FUNCTION_BLOCK ActivateTrackTask_TestSuite
VAR
	SetVelo AT%Q* : LREAL;
	AxisStatusFeedback AT%Q* : DWORD;
	stubAxis : AXIS_REF;
	stubTrack : XtsTrack('');
	testActivateTask : ActivateTrackTask := (AxisRef := stubAxis);
	TestSequence : INT;
	ThisTestSuite : TestSuite<TestSuiteParameter.MaxTestCount>('C:\ProgramData\Beckhoff\TwinCAT\3.1\Boot\ActiveTrack_Tests.xml') := (TestSuiteName := 'ActiveTrack Test Suite');
END_VAR

CASE TestSequence OF
	0: 
		SetVelo := 1.0;
		AxisStatusFeedback := 16#02100085;
		IF stubAxis.NcToPlc.SetVelo = 1.0 THEN
			TestSequence := 1;
		END_IF
	1:
		TaskRejectsCommandsWithNoAxis_Test();
		TaskRejectsDuplicateCommand_Test();
		TaskRejectsNullTrackCommand_Test();
		TaskRejectsCommandsIfAxisMoving_Test();
		TestSequence := 2;
	2:
		SetVelo := 0.0;
		IF stubAxis.NcToPlc.SetVelo = 0.0 THEN
			TestSequence := 3;
		END_IF
	3:
		TaskAcceptsCommand_Test();
		TestSequence := 4;
	4:
		AxisStatusFeedback := 16#00;
		IF stubAxis.Status.Disabled THEN
			TestSequence := 5;
		END_IF
	5:
		TaskRejectsCommandIfAxisDisabled_Test();
		TestSequence := 0;
END_CASE

stubAxis.ReadStatus();

METHOD TaskAcceptsCommand_Test
VAR_INST
	Expected : BOOL := TRUE;
	Actual	 : BOOL;
END_VAR
IF ThisTestSuite.Test(__POUNAME()).ExecuteTest() THEN
	Actual := SUCCEEDED(testActivateTask.Execute(Track := stubTrack));
	testActivateTask.Abort();
	ThisTestSuite.Test(__POUNAME()).AssertEqual(Expected, Actual);
END_IF
END_METHOD

METHOD TaskRejectsCommandIfAxisDisabled_Test
VAR_INST
	Expected : BOOL := TRUE;
	Actual	 : BOOL;
END_VAR
IF ThisTestSuite.Test(__POUNAME()).ExecuteTest() THEN
	//stubAxis.Status.Disabled := FALSE;
	Actual := FAILED(testActivateTask.Execute(Track := stubTrack));
	testActivateTask.Abort();
	ThisTestSuite.Test(__POUNAME()).AssertEqual(Expected, Actual);
END_IF
END_METHOD

METHOD TaskRejectsCommandsIfAxisMoving_Test
VAR_INST
	Expected : BOOL := TRUE;
	Actual	 : BOOL;
END_VAR
IF ThisTestSuite.Test(__POUNAME()).ExecuteTest() THEN
	Actual := FAILED(testActivateTask.Execute(Track := stubTrack));
	testActivateTask.Abort();
	ThisTestSuite.Test(__POUNAME()).AssertEqual(Expected, Actual);
END_IF
END_METHOD

METHOD TaskRejectsCommandsWithNoAxis_Test
VAR_INST
	Expected : BOOL := TRUE;
	Actual	 : BOOL;
END_VAR
IF ThisTestSuite.Test(__POUNAME()).ExecuteTest() THEN
	testActivateTask.AxisRef REF= 16#0;
	Actual := FAILED(testActivateTask.Execute(Track := stubTrack));
	testActivateTask.Abort();
	testActivateTask.AxisRef REF= stubAxis;
	ThisTestSuite.Test(__POUNAME()).AssertEqual(Expected, Actual);
END_IF
END_METHOD

METHOD TaskRejectsDuplicateCommand_Test
VAR_INST
	Expected : BOOL := TRUE;
	Actual	 : BOOL;
END_VAR
IF ThisTestSuite.Test(__POUNAME()).ExecuteTest() THEN
	testActivateTask.Execute(Track := stubTrack);
	Actual := FAILED(testActivateTask.Execute(Track := stubTrack));
	testActivateTask.Abort();
	ThisTestSuite.Test(__POUNAME()).AssertEqual(Expected, Actual);
END_IF
END_METHOD

METHOD TaskRejectsNullTrackCommand_Test
VAR_INST
	Expected : BOOL := TRUE;
	Actual	 : BOOL;
END_VAR
IF ThisTestSuite.Test(__POUNAME()).ExecuteTest() THEN
	Actual := FAILED(testActivateTask.Execute(Track := 16#0));
	testActivateTask.Abort();
	ThisTestSuite.Test(__POUNAME()).AssertEqual(Expected, Actual);
END_IF
END_METHOD

END_FUNCTION_BLOCK

(* stored: Version 1.1.0.1
   POU ActivateTrackTask_TestSuite: Id {433ac03a-1058-45df-bdb1-c68a454a01bf}, SpecialFunc None
   Method TaskAcceptsCommand_Test: Id {f38ea97e-61d4-4314-a23a-9dbdc22547e6}
   Method TaskRejectsCommandIfAxisDisabled_Test: Id {674d74d7-adee-4c2c-bfe4-b0e55b152e6f}
   Method TaskRejectsCommandsIfAxisMoving_Test: Id {892b298f-17bb-47e1-aafd-7aa4cff3908c}
   Method TaskRejectsCommandsWithNoAxis_Test: Id {d94842dc-f2af-4120-92da-d5763bf7c624}
   Method TaskRejectsDuplicateCommand_Test: Id {09fd1bc0-99f9-465b-899a-d4b787d799cb}
   Method TaskRejectsNullTrackCommand_Test: Id {f20a193c-f923-4de9-a85a-3ad1f9005177} *)
